FUNCTION_BLOCK AdsSocket
VAR_OUTPUT
	readBusy, readErr : BOOL;
	readErrId : UDINT;
	
	writeBusy, writeErr : BOOL;
	writeErrId : UDINT;
END_VAR
VAR_STAT
	localPrgName : STRING;
	localNetId : STRING;
	localPort : UINT;
END_VAR
VAR
	remotePrgName : STRING;
	remoteNetId : STRING;
	remotePort : UINT;
	
	adsReadSymbol : FB_ReadAdsSymByName;
	adsWriteSymbol : FB_WriteAdsSymByName;
END_VAR

METHOD close : BOOL
remotePrgName := '';
remoteNetId := '';
remotePort := 0;

//MEMSET(THIS, 0, SIZEOF(THIS^));
END_METHOD

METHOD open : BOOL
VAR_INPUT
	newLocalPrgName : STRING;
	newLocalNetId : T_AmsNetId;
	newLocalPort : T_AmsPort;
END_VAR
localPrgName := newLocalPrgName;
localNetId := newLocalNetId;
localPort := newLocalPort;
END_METHOD

METHOD read : BOOL
VAR_INPUT
	symbol : STRING;
	buffer : PVOID;
	symbolSize : UDINT;
END_VAR
adsReadSymbol.bRead := NOT adsReadSymbol.bRead;

adsReadSymbol(
	bRead:= , 
	sNetId:= remoteNetId, 
	nPort:= remotePort, 
	sVarName:= symbol, 
	nDestAddr:= buffer, 
	nLen:= symbolSize, 
	tTimeout:= , 
	eComMode:= , 
	bClearOnError:= TRUE, 
	bBusy=> readBusy,
	bError=> readErr, 
	nErrorId=> readErrId);
	
adsReadSymbol.bRead := FALSE;

read := NOT adsReadSymbol.bBusy AND NOT adsReadSymbol.bError;
END_METHOD

METHOD write : BOOL
VAR_INPUT
	symbol : STRING;
	data : PVOID;
	dataSize : UDINT;
END_VAR
adsWriteSymbol.bWrite := NOT adsWriteSymbol.bWrite;

adsWriteSymbol(
	bWrite:= , 
	sNetId:= remoteNetId, 
	nPort:= remotePort, 
	sVarName:= symbol, 
	nSrcAddr:= data, 
	nLen:= dataSize, 
	tTimeout:= , 
	eComMode:= , 
	bBusy=> , 
	bError=> , 
	nErrorId=> );
	
adsWriteSymbol.bWrite := FALSE;

write := NOT adsWriteSymbol.bBusy AND NOT adsWriteSymbol.bError;
END_METHOD

END_FUNCTION_BLOCK

(* stored: Version 1.1.0.1, ProductVersion 3.1.4024.11
   POU AdsSocket: Id {94b06c8f-6363-4f38-8057-d0f2ec092ac9}, SpecialFunc None
   Method close: Id {5b9b3a4a-f4db-4662-8e31-880b17578695}
   Method open: Id {41dcc539-006b-4672-ab53-559a081cb5fc}
   Method read: Id {76310918-f166-49dc-9eaa-fa797266bfbf}
   Method write: Id {78b7348b-168f-4aaf-82b1-6907845ef997} *)
